Staubli VAL3: makeTraj.pgx

public program makeTraj(string& x_sItem[])
  local num i
  local num l_nSize
  local tool l_tTool
  local bool l_bUnreached
  local point l_pPoint[2]
  local num l_nMoveId
  local bool l_bOk
  local ActionItem l_aAction
  local num j
  local TrajectoryItem l_tTraj
  local num l_nDistance
  local joint l_jJoint
  local Trajectory l_tTrajectory
begin
  //
  // inizialize the system
  //
  // take the TOOL
  call tcp:getTool(l_tTool,pt:tTraj[sTrajCycle].nIndexTool)
  //
  // for all of my traj cycleJoint move the robot
  //
  // the maximum size
  call getSizeItem(true,l_nSize)
  //
  // for all of my traj cyclePoints move the robot
  //
  resize(tTraj.tSuper,1,size(pt:tTraj[sTrajCycle].tData))
  for i=0 to (l_nSize-1)
    tTraj.tSuper[i]=pt:tTraj[sTrajCycle].tData[i].tSuper
  endFor
  tTraj.sID="JPOINT "+pt:tTraj[sTrajCycle].sID
  call cycleStatus:addTraj(tTraj)
  for i=0 to (l_nSize-1)
    //
    // get the point info
    //
    l_tTraj=pt:tTraj[sTrajCycle].tData[i].tSuper
    //
    // get the distance in percentage
    //
    call getDistance(l_tTool,l_nDistance,true,i)
    //
    // give to the traj library the percentage distance
    //
    if l_tTraj.toStop
      l_tTraj.nom_speed.blend=off
    endIf
    //
    // put the move in the stack
    //
    l_jJoint=pt:tTraj[sTrajCycle].tData[i].jJoint
    call moveTo(l_tTool,l_tTraj.nom_speed,l_tTraj.moveType,l_bUnreached,l_jJoint,l_nMoveId)
    // set the data
    l_aAction.nDistance=l_nDistance
    l_aAction.nPointId=i
    l_aAction.nMoveId=l_nMoveId
    l_aAction.sIdTraj="JPOINT "+pt:tTraj[sTrajCycle].sID
    call cycleStatus:putInstr_Traj(l_aAction,l_tTraj,pt:tTraj[sTrajCycle].nIndexTool,l_nSize)
    // there is a waitEndMove
    if l_tTraj.toStop
      waitEndMove()
      delay(l_tTraj.nStop)
      // wait all the action has been done
      wait(cycleStatus:bActionRunning==false)
    endIf
  endFor
end
